% RSLogix 500 project DIGITAL ROTAMETER FLOW CALCULATION.RSS, saved by version 8.30.00.16 %
PROJECT "SIM_PLC"    % processor: Bul.1763 MicroLogix 1100 Series B %

PROGRAM FILES
  LAD 2 "MAIN"  3 rungs
  LAD 3 "ROTAMETER"  3 rungs
  LAD 4 "CTRL LOGIC"  3 rungs

DATA FILES
  O0 OUTPUT  4 elements
  I1 INPUT  6 elements
  S2 STATUS  66 elements
  B3 BINARY  1 elements
  T4 TIMER  3 elements
  C5 COUNTER  1 elements
  R6 CONTROL  1 elements
  N7 INTEGER  1 elements
  F8 FLOAT  3 elements

LADDER 2 "MAIN"
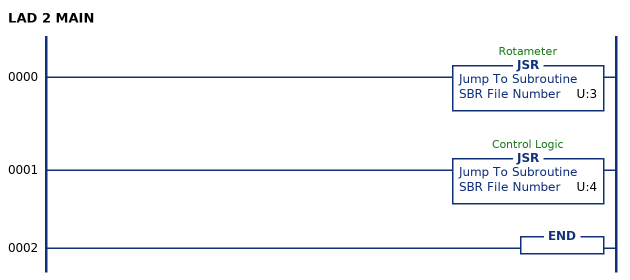
% Rung: 0 %
SOR JSR U:3 EOR
%   U:3  "Rotameter" %
% Rung: 1 %
SOR JSR U:4 EOR
%   U:4  "Control Logic" %
% Rung: 2 %
SOR END EOR

LADDER 3 "ROTAMETER"
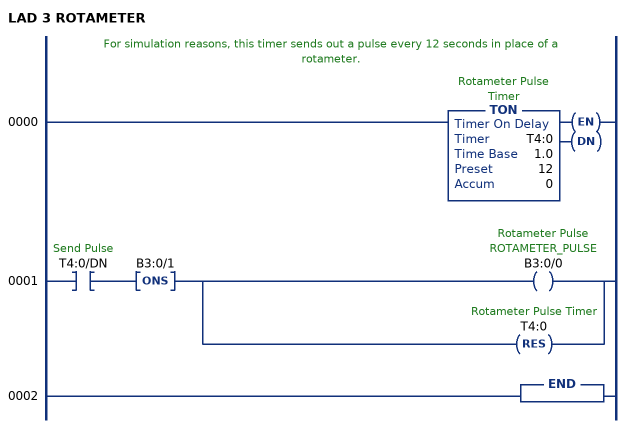
% Rung: 0 %
% For simulation reasons, this timer sends out a pulse every 12 seconds in place of a rotameter. %
SOR TON T4:0 1.0 12 0 EOR
%   T4:0  "Rotameter Pulse Timer" %
% Rung: 1 %
SOR XIC T4:0/DN ONS B3:0/1 BST OTE B3:0/0 NXB RES T4:0 BND EOR
%   T4:0/DN  "Send Pulse" %
%   B3:0/0  ROTAMETER_PULSE  "Rotameter Pulse" %
%   T4:0  "Rotameter Pulse Timer" %
% Rung: 2 %
SOR END EOR

LADDER 4 "CTRL LOGIC"
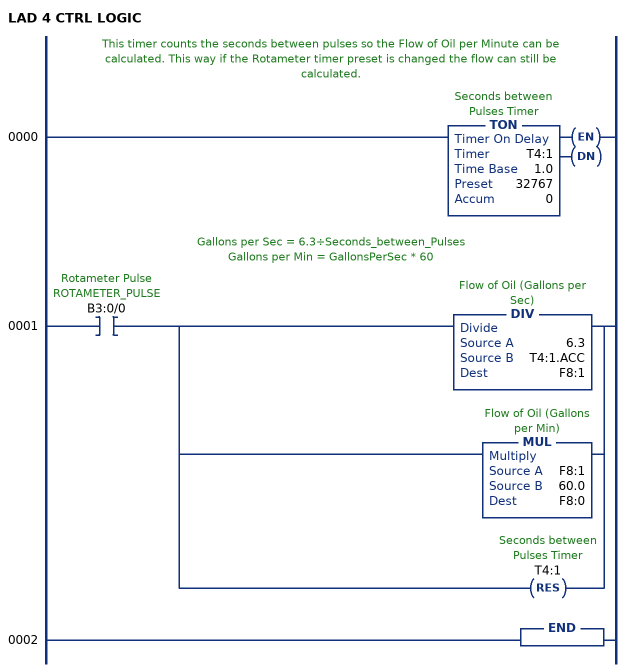
% Rung: 0 %
% This timer counts the seconds between pulses so the Flow of Oil per Minute can be calculated. This way if the Rotameter timer preset is changed the flow can still be calculated. %
SOR TON T4:1 1.0 32767 0 EOR
%   T4:1  "Seconds between Pulses Timer" %
% Rung: 1 %
% Gallons per Sec = 6.3÷Seconds_between_Pulses
% 
% Gallons per Min = GallonsPerSec * 60 %
SOR XIC B3:0/0 BST DIV 6.3 T4:1.ACC F8:1 NXB MUL F8:1 60.0 F8:0 NXB RES T4:1 BND EOR
%   B3:0/0  ROTAMETER_PULSE  "Rotameter Pulse" %
%   T4:1.ACC  "Seconds Between Pulses" %
%   F8:1  "Flow of Oil (Gallons per Sec)" %
%   F8:0  "Flow of Oil (Gallons per Min)" %
%   T4:1  "Seconds between Pulses Timer" %
% Rung: 2 %
SOR END EOR

OTHER DOCUMENTED ADDRESSES
  C5:0.ACC  "Pulses per Minute"

DATA TABLE (non-zero values as saved)
DATA T4
% .PRE .ACC %
% T4:0 % 12 0
% T4:1 % 32767 0
% T4:2 % 60 0
DATA C5
% .PRE .ACC %
% C5:0 % 32767 0
